INTERFACE I_TestComponent EXTENDS I_BaseFB

END_INTERFACE

(* stored: Version 1.1.0.1
   Itf I_TestComponent: Id {ca947f9d-2dd4-42c6-a605-220dd9999fff} *)
